TYPE "UDT_SUCActiveElement"
VERSION : 0.1
   STRUCT
      tag_name : String;
      tag_description : String;
      OSLevel : Int;
      WQC : Int;
   END_STRUCT;

END_TYPE

